FUNCTION_BLOCK RingTokenConveyerCTL (* Composite Function Block Type *)
  (* Standard: 61499-2 *)
  (* Version 0.2, 2003-12-05, JHC, Rockwell Automation, Renamed from NEWCOMPFB. *)
  (* Version 0.1, 2002-01-08, JHC, Rockwell Automation, Added DLY FB as example. *)
  (* Version 0.0, 2000-05-27, JHC, Rockwell Automation *)
  (* Compiler header: package fb.rt.cs725; *)
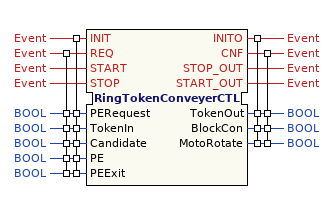
  EVENT_INPUT
    INIT WITH PERequest, TokenIn, PE, Candidate, PEExit; (* Initialization Request *)
    REQ WITH PERequest, TokenIn, Candidate, PE, PEExit; (* Normal Execution Request *)
    START;
    STOP;
  END_EVENT
  EVENT_OUTPUT
    INITO WITH TokenOut, MotoRotate, BlockCon; (* Initialization Confirm *)
    CNF WITH TokenOut, BlockCon, MotoRotate; (* Execution Confirmation *)
    STOP_OUT;
    START_OUT;
  END_EVENT
  VAR_INPUT
    PERequest : BOOL; (* Input event qualifier *)
    TokenIn : BOOL;
    Candidate : BOOL;
    PE : BOOL;
    PEExit : BOOL;
  END_VAR
  VAR_OUTPUT
    TokenOut : BOOL;
    BlockCon : BOOL;
    MotoRotate : BOOL;
  END_VAR
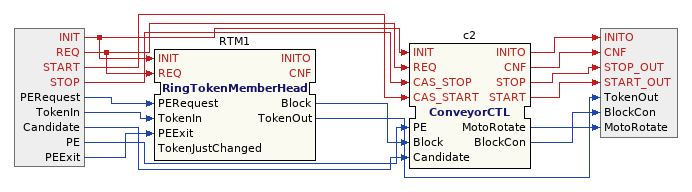
  FBS
    RTM1 : RingTokenMemberHead;
    c2 : ConveyorCTL;
  END_FBS
  EVENT_CONNECTIONS
    INIT TO RTM1.INIT;
    REQ TO RTM1.REQ;
    c2.START TO START_OUT;
    c2.STOP TO STOP_OUT;
    c2.CNF TO CNF;
    c2.INITO TO INITO;
    INIT TO c2.INIT;
    REQ TO c2.REQ;
    STOP TO c2.CAS_STOP;
    START TO c2.CAS_START;
  END_CONNECTIONS
  DATA_CONNECTIONS
    c2.MotoRotate TO MotoRotate;
    c2.BlockCon TO BlockCon;
    RTM1.TokenOut TO TokenOut;
    TokenIn TO RTM1.TokenIn;
    PE TO c2.PE;
    Candidate TO c2.Candidate;
    PERequest TO RTM1.PERequest;
    RTM1.Block TO c2.Block;
    PEExit TO RTM1.PEExit;
  END_CONNECTIONS
END_FUNCTION_BLOCK
